// TIA Portal V18 export
FUNCTION_BLOCK "Planta"   // FB2, LAD
{ S7_Optimized_Access := 'FALSE' }
// stored: SetENOAutomatically false
   VAR_INPUT
      Valve : Bool;
      PID_output : Real;
   END_VAR
   VAR_OUTPUT
      Physvar : Real;
   END_VAR
   VAR
      F1 : Bool;
      F2 : Bool;
      F3 : Bool;
      F4 : Bool;
      F5 : Bool;
      F6 : Bool;
      LL : Real := 20.0;
      L : Real := 40.0;
      H : Real := 60.0;
      HH : Real := 80.0;
      LL_M : Real := 0.01;
      L_M : Real := 0.05;
      H_M : Real := 0.1;
      HH_M : Real := 0.2;
      MAX_M : Real := 0.5;
      Out_M : Real := 0.1;
   END_VAR
   VAR_TEMP   // added for the SCL form of the ladder/FBD networks
      _w1 : Bool;
   END_VAR
BEGIN

REGION Network 1
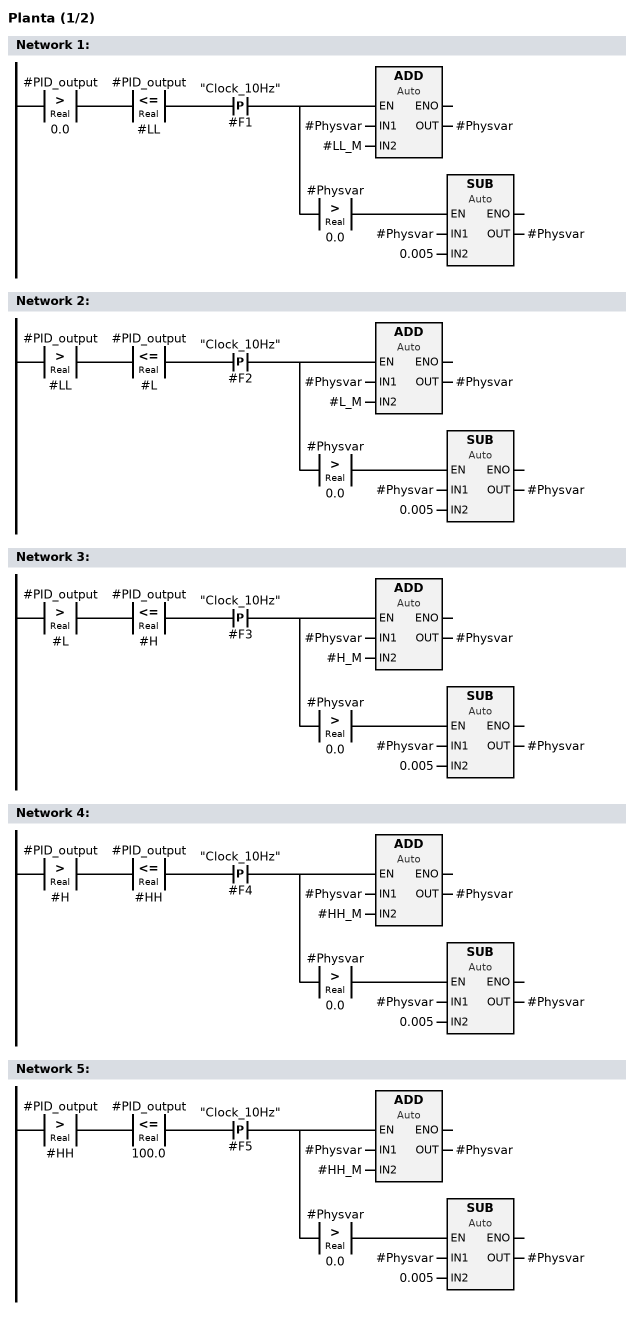
   RUNG wire#powerrail
      { S7_Templates := "SrcType := Real" } GT_Contact(in1 := #PID_output, in2 := 0.0)
      { S7_Templates := "SrcType := Real" } LE_Contact(in1 := #PID_output, in2 := #LL)
      P_Contact(operand := "Clock_10Hz", bit := #F1)
      wire#w1
      Add(in1 := #Physvar, in2 := #LL_M, out => #Physvar)
   END_RUNG
   RUNG wire#w1
      { S7_Templates := "SrcType := Real" } GT_Contact(in1 := #Physvar, in2 := 0.0)
      Sub(in1 := #Physvar, in2 := 0.005, out => #Physvar)
   END_RUNG
   // the same network as SCL:
   #_w1 := (#PID_output > 0.0) AND (#PID_output <= #LL) AND "Clock_10Hz" AND NOT #F1;   // rising edge of "Clock_10Hz"
   #F1 := "Clock_10Hz";
   IF #_w1 THEN #Physvar := #Physvar + #LL_M; END_IF;
   IF #_w1 AND (#Physvar > 0.0) THEN #Physvar := #Physvar - 0.005; END_IF;
END_REGION

REGION Network 2
   RUNG wire#powerrail
      { S7_Templates := "SrcType := Real" } GT_Contact(in1 := #PID_output, in2 := #LL)
      { S7_Templates := "SrcType := Real" } LE_Contact(in1 := #PID_output, in2 := #L)
      P_Contact(operand := "Clock_10Hz", bit := #F2)
      wire#w1
      Add(in1 := #Physvar, in2 := #L_M, out => #Physvar)
   END_RUNG
   RUNG wire#w1
      { S7_Templates := "SrcType := Real" } GT_Contact(in1 := #Physvar, in2 := 0.0)
      Sub(in1 := #Physvar, in2 := 0.005, out => #Physvar)
   END_RUNG
   // the same network as SCL:
   #_w1 := (#PID_output > #LL) AND (#PID_output <= #L) AND "Clock_10Hz" AND NOT #F2;   // rising edge of "Clock_10Hz"
   #F2 := "Clock_10Hz";
   IF #_w1 THEN #Physvar := #Physvar + #L_M; END_IF;
   IF #_w1 AND (#Physvar > 0.0) THEN #Physvar := #Physvar - 0.005; END_IF;
END_REGION

REGION Network 3
   RUNG wire#powerrail
      { S7_Templates := "SrcType := Real" } GT_Contact(in1 := #PID_output, in2 := #L)
      { S7_Templates := "SrcType := Real" } LE_Contact(in1 := #PID_output, in2 := #H)
      P_Contact(operand := "Clock_10Hz", bit := #F3)
      wire#w1
      Add(in1 := #Physvar, in2 := #H_M, out => #Physvar)
   END_RUNG
   RUNG wire#w1
      { S7_Templates := "SrcType := Real" } GT_Contact(in1 := #Physvar, in2 := 0.0)
      Sub(in1 := #Physvar, in2 := 0.005, out => #Physvar)
   END_RUNG
   // the same network as SCL:
   #_w1 := (#PID_output > #L) AND (#PID_output <= #H) AND "Clock_10Hz" AND NOT #F3;   // rising edge of "Clock_10Hz"
   #F3 := "Clock_10Hz";
   IF #_w1 THEN #Physvar := #Physvar + #H_M; END_IF;
   IF #_w1 AND (#Physvar > 0.0) THEN #Physvar := #Physvar - 0.005; END_IF;
END_REGION

REGION Network 4
   RUNG wire#powerrail
      { S7_Templates := "SrcType := Real" } GT_Contact(in1 := #PID_output, in2 := #H)
      { S7_Templates := "SrcType := Real" } LE_Contact(in1 := #PID_output, in2 := #HH)
      P_Contact(operand := "Clock_10Hz", bit := #F4)
      wire#w1
      Add(in1 := #Physvar, in2 := #HH_M, out => #Physvar)
   END_RUNG
   RUNG wire#w1
      { S7_Templates := "SrcType := Real" } GT_Contact(in1 := #Physvar, in2 := 0.0)
      Sub(in1 := #Physvar, in2 := 0.005, out => #Physvar)
   END_RUNG
   // the same network as SCL:
   #_w1 := (#PID_output > #H) AND (#PID_output <= #HH) AND "Clock_10Hz" AND NOT #F4;   // rising edge of "Clock_10Hz"
   #F4 := "Clock_10Hz";
   IF #_w1 THEN #Physvar := #Physvar + #HH_M; END_IF;
   IF #_w1 AND (#Physvar > 0.0) THEN #Physvar := #Physvar - 0.005; END_IF;
END_REGION

REGION Network 5
   RUNG wire#powerrail
      { S7_Templates := "SrcType := Real" } GT_Contact(in1 := #PID_output, in2 := #HH)
      { S7_Templates := "SrcType := Real" } LE_Contact(in1 := #PID_output, in2 := 100.0)
      P_Contact(operand := "Clock_10Hz", bit := #F5)
      wire#w1
      Add(in1 := #Physvar, in2 := #HH_M, out => #Physvar)
   END_RUNG
   RUNG wire#w1
      { S7_Templates := "SrcType := Real" } GT_Contact(in1 := #Physvar, in2 := 0.0)
      Sub(in1 := #Physvar, in2 := 0.005, out => #Physvar)
   END_RUNG
   // the same network as SCL:
   #_w1 := (#PID_output > #HH) AND (#PID_output <= 100.0) AND "Clock_10Hz" AND NOT #F5;   // rising edge of "Clock_10Hz"
   #F5 := "Clock_10Hz";
   IF #_w1 THEN #Physvar := #Physvar + #HH_M; END_IF;
   IF #_w1 AND (#Physvar > 0.0) THEN #Physvar := #Physvar - 0.005; END_IF;
END_REGION

REGION Network 6
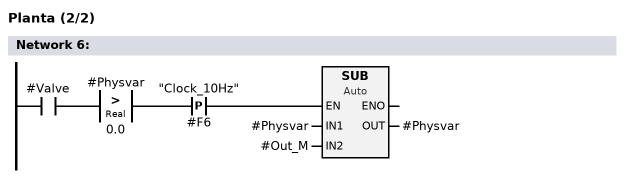
   RUNG wire#powerrail
      Contact( #Valve )
      { S7_Templates := "SrcType := Real" } GT_Contact(in1 := #Physvar, in2 := 0.0)
      P_Contact(operand := "Clock_10Hz", bit := #F6)
      Sub(in1 := #Physvar, in2 := #Out_M, out => #Physvar)
   END_RUNG
   // the same network as SCL:
   #_w1 := #Valve AND (#Physvar > 0.0) AND "Clock_10Hz" AND NOT #F6;   // rising edge of "Clock_10Hz"
   #F6 := "Clock_10Hz";
   IF #_w1 THEN #Physvar := #Physvar - #Out_M; END_IF;
END_REGION
END_FUNCTION_BLOCK
